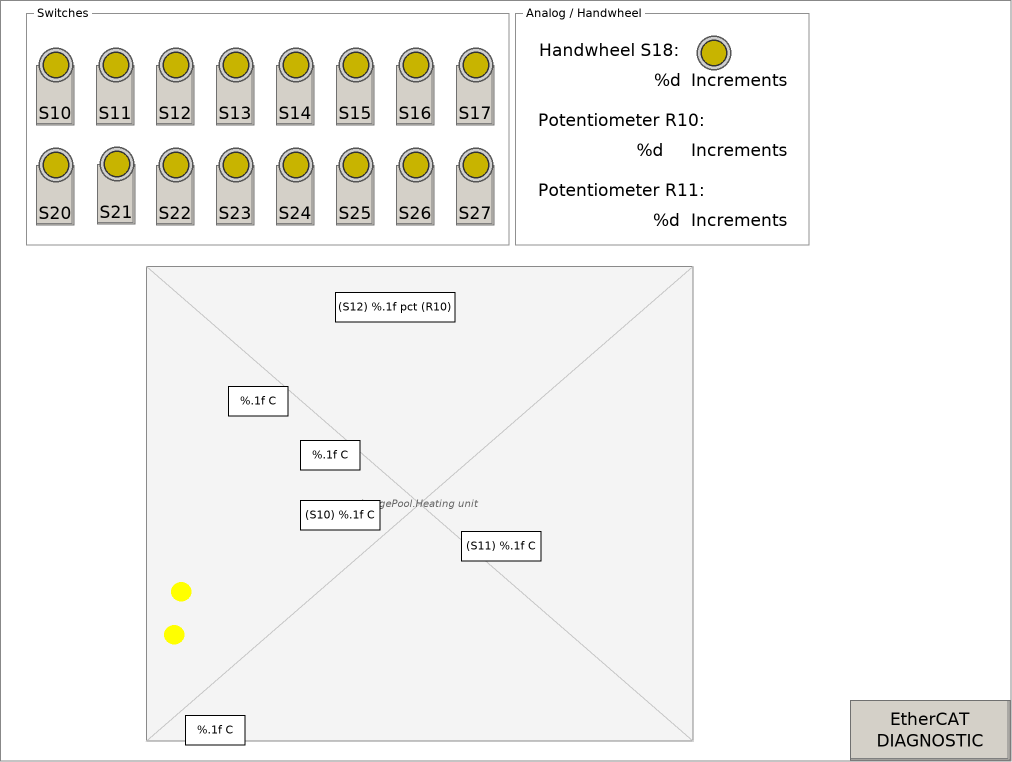
VISUALIZATION HmiStartPage  // 1012x762
    Image (146,266 547x475), image: ImagePool.Heating unit
    Button (850,700 160x60), "EtherCAT DIAGNOSTIC"
        OnMouseClick: change screen: HmiEtherCatDiagnostic
    GroupBox (26,5 483x240), "Switches"
        Button (10,60 38x60), "S10", colour toggle: bSwitchS10
            toggle bSwitchS10
        Lamp1 (10,40 40x40), variable: bLedH10, style: Lamp-Lamp1-Yellow
        Button (70,60 38x60), "S11", colour toggle: bSwitchS11
            toggle bSwitchS11
        Lamp1 (70,40 40x40), variable: bLedH11, style: Lamp-Lamp1-Yellow
        Button (130,60 38x60), "S12", colour toggle: bSwitchS12
            toggle bSwitchS12
        Lamp1 (130,40 40x40), variable: bLedH12, style: Lamp-Lamp1-Yellow
        Button (190,60 38x60), "S13", colour toggle: bSwitchS13
            toggle bSwitchS13
        Lamp1 (190,40 40x40), variable: bLedH13, style: Lamp-Lamp1-Yellow
        Button (250,60 38x60), "S14", colour toggle: bSwitchS14
            toggle bSwitchS14
        Lamp1 (250,40 40x40), variable: bLedH14, style: Lamp-Lamp1-Yellow
        Button (310,60 38x60), "S15", colour toggle: bSwitchS15
            toggle bSwitchS15
        Lamp1 (310,40 40x40), variable: bLedH15, style: Lamp-Lamp1-Yellow
        Button (370,60 38x60), "S16", colour toggle: bSwitchS16
            toggle bSwitchS16
        Lamp1 (370,40 40x40), variable: bLedH16, style: Lamp-Lamp1-Yellow
        Button (430,60 38x60), "S17", colour toggle: bSwitchS17
            toggle bSwitchS17
        Lamp1 (430,40 40x40), variable: bLedH17, style: Lamp-Lamp1-Yellow
        Button (10,160 38x60), "S20", colour toggle: bSwitchS20
            toggle bSwitchS20
        Lamp1 (10,140 40x40), variable: bLedH20, style: Lamp-Lamp1-Yellow
        Button (71,159 38x60), "S21", colour toggle: bSwitchS21
            toggle bSwitchS21
        Lamp1 (71,139 40x40), variable: bLedH21, style: Lamp-Lamp1-Yellow
        Button (130,160 38x60), "S22", colour toggle: bSwitchS22
            toggle bSwitchS22
        Lamp1 (130,140 40x40), variable: bLedH22, style: Lamp-Lamp1-Yellow
        Button (190,160 38x60), "S23", colour toggle: bSwitchS23
            toggle bSwitchS23
        Lamp1 (190,140 40x40), variable: bLedH23, style: Lamp-Lamp1-Yellow
        Button (250,160 38x60), "S24", colour toggle: bSwitchS24
            toggle bSwitchS24
        Lamp1 (250,140 40x40), variable: bLedH24, style: Lamp-Lamp1-Yellow
        Button (310,160 38x60), "S25", colour toggle: bSwitchS25
            toggle bSwitchS25
        Lamp1 (310,140 40x40), variable: bLedH25, style: Lamp-Lamp1-Yellow
        Button (370,160 38x60), "S26", colour toggle: bSwitchS26
            toggle bSwitchS26
        Lamp1 (370,140 40x40), variable: bLedH26, style: Lamp-Lamp1-Yellow
        Button (430,160 38x60), "S27", colour toggle: bSwitchS27
            toggle bSwitchS27
        Lamp1 (430,140 40x40), variable: bLedH27, style: Lamp-Lamp1-Yellow
    GroupBox (515,5 294x240), "Analog / Handwheel"
        Rectangle (20,200 148x30), "%d", text variable: nAnalogInR11
            OnMouseClick: write the text variable via Default, min 0, max 32767
        Label (173,200 118x30), "Increments"
        Label (20,170 197x30), "Potentiometer R11:"
        Rectangle (20,130 148x30), "%d", text variable: nAnalogInR10
            OnMouseClick: write the text variable via Default, min 0, max 32767
        Label (173,130 121x30), "Increments"
        Label (20,100 216x30), "Potentiometer R10:"
        Lamp1 (179,28 40x40), variable: bHandwheelSwitchS18, style: Lamp-Lamp1-Yellow
        Rectangle (21,60 148x30), "%d", text variable: nHandwheelCounter
            OnMouseClick: write the text variable via Default
        Label (173,60 133x30), "Increments"
        Label (21,30 216x30), "Handwheel S18:"
    Rectangle (300,500 80x30), "(S10) %.1f C", text variable: TemperatureControl.fTemperatureCHeating1, colour toggle: bHeating1Aktiv
    Rectangle (461,531 80x30), "(S11) %.1f C", text variable: TemperatureControl.fTemperatureCHeating2, colour toggle: bHeating2Aktiv
    Rectangle (300,440 60x30), "%.1f C", text variable: TemperatureControl.fTemperatureCHeatSink
    Rectangle (228,386 60x30), "%.1f C", text variable: TemperatureControl.fTemperatureCCoverHeating
    Rectangle (185,715 60x30), "%.1f C", text variable: TemperatureControl.fTemperatureCAmbient
    Rectangle (335,292 120x30), "(S12) %.1f pct (R10)", text variable: TemperatureControl.fVeloFanProcent, colour toggle: nFanStatus.1
    Ellipse (171,582 20x19), invisible if: NOT bHeating1Led
    Ellipse (164,625 20x19), invisible if: NOT bHeating2Led
END_VISUALIZATION

(* stored: Version 1.1.0.1
   Visu HmiStartPage: Id {81da00b4-351b-4bea-beba-4843bfdabd99} *)
